# EPICS IOC start-up script: require/3.1.2/siteMods/mrfioc2/2.2.1rc3/iocrc.iocsh
require "supercycleEngine" "1.0.0rc8"
require "mrfioc2" "2.2.1rc3"
epicsEnvSet "PEVG" "TD-M:Ctrl-EVG-1"
epicsEnvSet "PSCE" "TD-M:Ctrl-SCE-1"
epicsEnvSet "PCI_SLOT" "0e:00.0"
epicsEnvSet "reftabs_DIR" "/opt/reftabs"
epicsEnvSet "ASYNARGS" "EvtPMortem=40, EvtPMortemSys=41, EvtDoD=42, EvtDoDSys=43"
